FUNCTION F_Time2lrSecond : lreal
VAR_INPUT
	t : TIME;
END_VAR
VAR
END_VAR

F_Time2lrSecond := time_to_lreal(t)/1000;

END_FUNCTION

(* stored: Version 1.1.0.1, ProductVersion 3.1.4024.12
   POU F_Time2lrSecond: Id {52b6d15b-b1cf-4e87-ae0e-f34c55f99025}, SpecialFunc None *)
